FUNCTION_BLOCK FB_SaMElementStopped EXTENDS FB_SaMElement
VAR
END_VAR

METHOD FB_init : BOOL
VAR_INPUT
	bInitRetains : BOOL; // if TRUE, the retain variables are initialized (warm start / cold start)
	bInCopyCode : BOOL;  // if TRUE, the instance afterwards gets moved into the copy code (online change)
END_VAR
THIS^.bTypeActive		:= FALSE;

THIS^.SetText (eLocation := E_BaseLocation.pl, wsDescription := "Zatrzymany");
THIS^.SetText (eLocation := E_BaseLocation.en, wsDescription := "Stopped");
THIS^.SetText (eLocation := E_BaseLocation.de, wsDescription := "Gestoppt");
THIS^.SetName (stName := THIS^.GetTexts ());
END_METHOD

METHOD PUBLIC InvokeStateForTopElement : BOOL
VAR_INPUT
	itfTopElement		: ITF_BaseSaMStateMethod;
END_VAR
InvokeStateForTopElement	:= itfTopElement.SP_Stopped ();
END_METHOD

END_FUNCTION_BLOCK

(* stored: Version 1.1.0.1
   POU FB_SaMElementStopped: Id {9d16f680-9f14-0072-25ae-30fba7085f68}, SpecialFunc None
   Method FB_init: Id {dbc34390-c6a1-021c-12c1-a13416849511}
   Method InvokeStateForTopElement: Id {774b14ad-3f8b-0124-09ec-de3eaa5ab2c7} *)
